// Mitsubishi GX Works2 project: 28-06-2Code mau   PLC: FX3G

PROGRAM MAIN
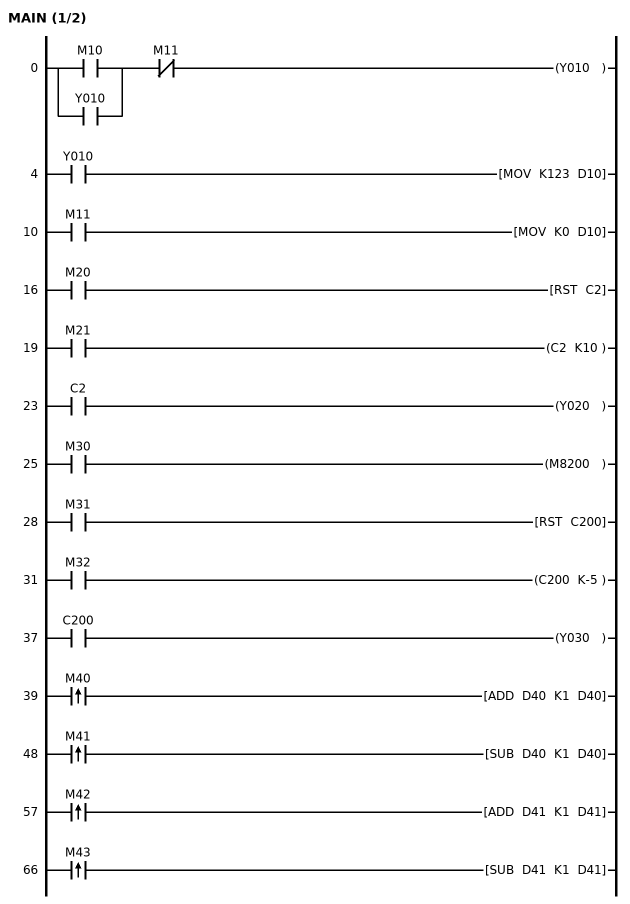
0     LD      M10
      OR      Y010
      ANI     M11
      OUT     Y010
4     LD      Y010
      MOV     K123 D10
10    LD      M11
      MOV     K0 D10
16    LD      M20
      RST     C2
19    LD      M21
      OUT     C2 K10
23    LD      C2
      OUT     Y020
25    LD      M30
      OUT     M8200
28    LD      M31
      RST     C200
31    LD      M32
      OUT     C200 K-5
37    LD      C200
      OUT     Y030
39    LDP     M40
      ADD     D40 K1 D40
48    LDP     M41
      SUB     D40 K1 D40
57    LDP     M42
      ADD     D41 K1 D41
66    LDP     M43
      SUB     D41 K1 D41
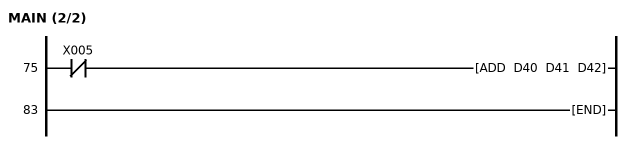
75    LDI     X005
      ADD     D40 D41 D42
83    END
END_PROGRAM
